(* PLC project Relay, NYU-AD Simple 1, author Marios Sazos *)
(* stored: creationDateTime 2017-09-06T16:00:31, version 1, modificationDateTime 2018-03-20T16:39:54 *)

PROGRAM Overcurrent
  VAR
    phase_1 AT %IX0.1 : BOOL;
  END_VAR
  VAR
    trip_fault : BOOL;
  END_VAR
  VAR
    phase_2 AT %IX0.2 : BOOL;
    phase_3 AT %IX0.3 : BOOL;
    local_trip AT %IX0.4 : BOOL;
    local_close AT %IX0.5 : BOOL;
    trip AT %QX0.7 : BOOL;
    close AT %QX0.6 : BOOL;
    remote_trip AT %QX0.0 : BOOL;
    remote_close AT %QX0.1 : BOOL;
    current_RMS AT %MW0 : UINT;
  END_VAR
  VAR
    ct_ratio : LINT := 1000;
    threshold : UINT := 300;
  END_VAR
  VAR
    I_RMS AT %IW0 : UINT;
  END_VAR
  VAR
    T1 : TOF;
    T2 : TON;
  END_VAR
  VAR  (* added by the conversion: wires and edge detectors of the diagram *)
    _LINT_TO_UINT48_OUT : UINT;
  END_VAR

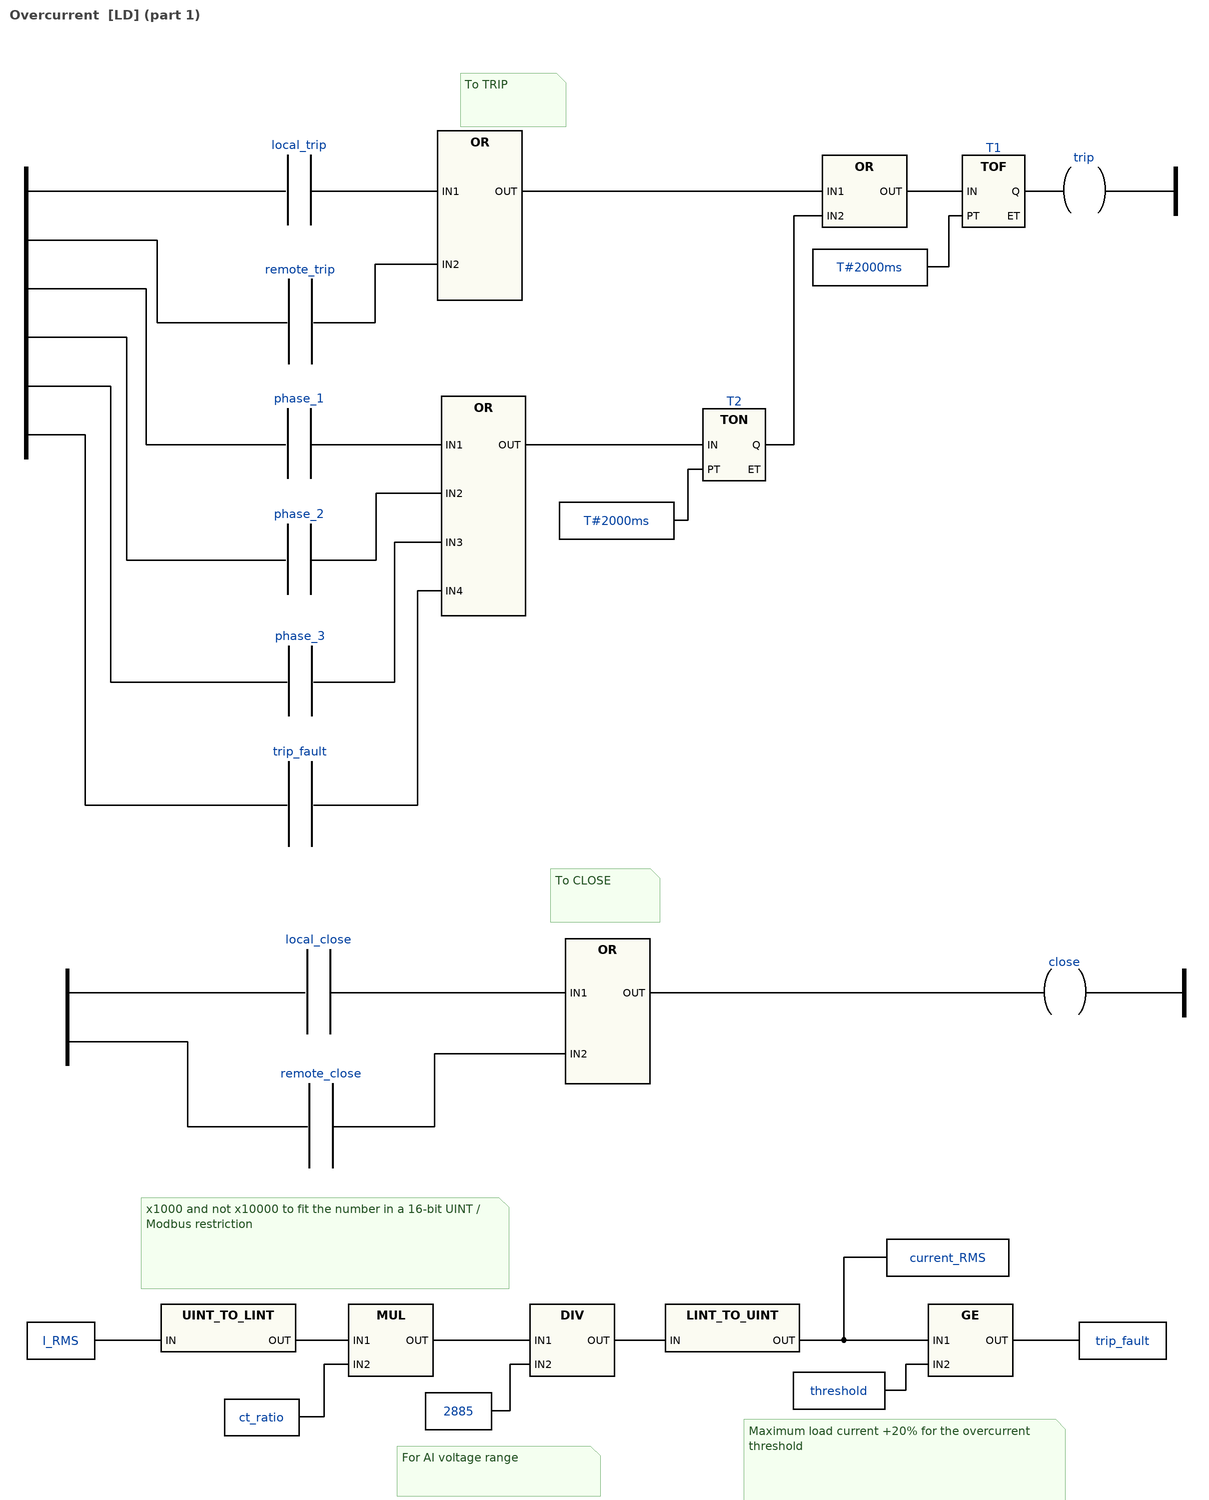
(* LD diagram, written out as Structured Text *)
(* To TRIP *)
T2(IN := phase_1 OR phase_2 OR phase_3 OR trip_fault, PT := T#2000ms);
T1(IN := local_trip OR remote_trip OR T2.Q, PT := T#2000ms);
trip := T1.Q;
(* To CLOSE *)
close := local_close OR remote_close;
(* x1000 and not x10000 to fit the number in a 16-bit UINT / Modbus restriction *)
_LINT_TO_UINT48_OUT := LINT_TO_UINT(UINT_TO_LINT(I_RMS) * ct_ratio / 2885);
current_RMS := _LINT_TO_UINT48_OUT;
trip_fault := _LINT_TO_UINT48_OUT >= threshold;
(* Maximum load current +20% for the overcurrent threshold *)
(* For AI voltage range *)
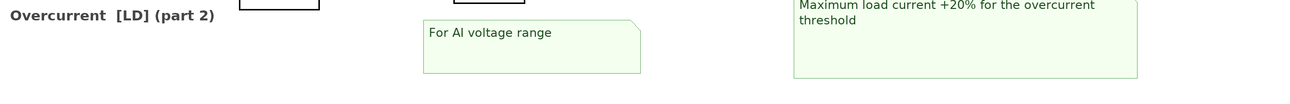
END_PROGRAM

CONFIGURATION Config0
  RESOURCE Res0 ON PLC
    TASK TaskMain(INTERVAL := T#50ms, PRIORITY := 0);
    PROGRAM Inst0 WITH TaskMain : Overcurrent;
  END_RESOURCE
END_CONFIGURATION
